// TwinCAT 3 PLC project TestProject
// ProgramVersion: 3.1.4026.24
// libraries:
//   Tc2_MC2, * (Beckhoff Automation GmbH)
//   Tc2_Standard, * (Beckhoff Automation GmbH)
//   Tc2_System, * (Beckhoff Automation GmbH)
// project tree:
//   / PlcTask.TcTTO
//   POUs/ AxisControl.TcPOU, MAIN.TcPOU
// real-time tasks:
//   TASK PlcTask: cycle T#10ms, priority 20, ADS port 350
// motion (NC):
//   TASK NC-Task 1 SAF: cycle T#2ms, priority 4, ADS port 501
//   TASK NC-Task 1 SVB: cycle T#10ms, priority 8, ADS port 511
//   AXIS Axis 1 (id 1)
//     General: UnitName=m
//     OtherSettings: AllowMotionCmdToSlave=true
//     encoder EncType=16
//       EncPara: MaxCount=#x0000ffff
//     drive DrvType=13
//       Analog: TorqueSetpointScale=10, ScaleFactorActTorque=0.1
//       TimeComp: TaskDelayCycles=1
//     controller CtrType=1
//       CtrPara: PriorControlFactor=1
//         Observer: BandWidth=20
// I/O:
//   DEVICE EtcMaster (EtherCAT), AmsNetId 192.168.1.10.2.1
//     Term 1 (EK1100) [EK1100 EtherCAT Coupler (2A E-Bus)]
//       Term 2 (EL1008) [EL1008 8Ch. Dig. Input 24V, 3ms]
//       Term 3 (EL2008) [EL2008 8Ch. Dig. Output 24V, 0.5A]
//       Term 4 (EL3443) [EL3443 3Ch. Power Measuring]
//       Term 5 (EL6224) [EL6224 (IO Link Master)]
//       Term 6 (EL1918) [EL1918, 8Ch. Safety Input 24V, TwinSAFE]
//         modules: Module 1 (FSOE), Module 2 (FSLOGIC)
//       Term 7 (EL9011) [EL9011 End Terminal]
// variable links:
//   (this object) <-> NC-Task 1 SAF/Axes/Axis 1
//     PlcTask Inputs/MAIN.Axis1.ax.NcToPlc <-> Outputs/ToPlc
//     PlcTask Outputs/MAIN.Axis1.ax.PlcToNc <-> Inputs/FromPlc

CONFIGURATION TestProject
    RESOURCE PLC ON TwinCAT3
        TASK PlcTask(INTERVAL := T#10ms, PRIORITY := 20);
        PROGRAM MAIN WITH PlcTask : MAIN;
    END_RESOURCE
END_CONFIGURATION

// ---- POUs/MAIN.TcPOU
PROGRAM MAIN
VAR
	Axis1		: AxisControl;
	
	PowerOn		: BOOL;
	ResetAxis	: BOOL;
	MoveAxis	: BOOL;
	StopAxis	: BOOL;
	AxisPos		: LREAL;
	Velocity	: LREAL := 0.1;
	AxisErrorID	: DWORD;
END_VAR

IF ResetAxis THEN
	ResetAxis := NOT Axis1.Reset();
ELSIF MoveAxis THEN
	MoveAxis := NOT Axis1.MoveAxis(Velocity:= Velocity);
ELSIF StopAxis THEN
	StopAxis := NOT Axis1.StopAxis();
END_IF

Axis1.PowerAxis(Enable:= PowerOn);
Axis1();
AxisPos := Axis1.Position;
AxisErrorID := Axis1.AxisError;

END_PROGRAM

// ---- POUs/AxisControl.TcPOU
FUNCTION_BLOCK AxisControl
VAR
	ax			: AXIS_REF;
	mcPower		: MC_Power;
	mcReset		: MC_Reset;
	mcMoveVel	: MC_MoveVelocity;
	mcHalt		: MC_Halt;
	
	_powerOn	: BOOL;
	_reset		: BOOL;
	_moveVel	: BOOL;
	_stop		: BOOL;
	_velocity	: LREAL;
END_VAR

ax.ReadStatus();

mcPower(Axis:= ax, Enable:= _powerOn, Enable_Positive:= _powerOn,	Enable_Negative:= _powerOn);

mcReset(Axis:= ax, Execute:= _reset);
IF mcReset.Done THEN
	mcReset(Axis:= ax, Execute:= FALSE);
	_reset := FALSE;
END_IF

mcMoveVel(Axis:= ax, Execute:= _moveVel, Velocity:= _velocity);
IF mcMoveVel.InVelocity THEN
	_moveVel := FALSE;
END_IF

mcHalt(Axis:= ax, Execute:= _stop);	
IF mcHalt.Done THEN
	_stop := FALSE;
END_IF

PROPERTY AxisError : DWORD
GET
AxisError := UDINT_TO_DWORD(ax.Status.ErrorID);
END_GET
END_PROPERTY

METHOD MoveAxis : BOOL
VAR_INPUT
	Velocity: LREAL := 0.1;
END_VAR
_moveVel := TRUE;
_stop := FALSE;
_velocity := Velocity;

MoveAxis := TRUE;
END_METHOD

PROPERTY Position : LREAL
GET
Position := ax.NcToPlc.ActPos;
END_GET
END_PROPERTY

METHOD PowerAxis : BOOL
VAR_INPUT
	Enable: BOOL;
END_VAR
_powerOn := Enable;

PowerAxis := TRUE;
END_METHOD

METHOD Reset : BOOL
_reset := TRUE;
_moveVel := FALSE;
_stop := FALSE;

Reset := TRUE;
END_METHOD

METHOD StopAxis : BOOL
_moveVel := FALSE;
_stop := TRUE;

StopAxis := TRUE;
END_METHOD

END_FUNCTION_BLOCK
